{attribute 'GeneratedUsingTerminal: EL3773-0000-0016'}
{attribute addProperty BoxType "EL3773-0000-0016"}
{attribute addProperty Id "U1_SAMPLESAT %I*U1_SAMPLES_2D13B74B20"}
{attribute addProperty CRC "3982986734"}
{attribute addProperty Size "20"}
TYPE L1_Voltage_Samples_ED678DEE :
STRUCT
	{attribute addProperty Name "U1_SAMPLES"}
	U1_SAMPLES AT %I* : U1_SAMPLES_2D13B74B;
END_STRUCT
END_TYPE
